TYPE DUT_SourceDataStore :
STRUCT
    {attribute 'pytmc' := 'pv: Valve'}
    fbSourceValve : REFERENCE TO FB_VGC;
    {attribute 'pytmc' := '
        pv: Valid
        io: input
        field: ZNAM Data Invalid
        field: ONAM Data Valid
        field: ZSV MAJOR
        field: OSV NO_ALARM
    '}
    bDataValid : BOOL;

    {attribute 'pytmc' := '
        pv: ChecksOK
        io: input
        field: ZNAM Failed
        field: ONAM Passed
        field: ZSV MAJOR
        field: OSV NO_ALARM
    '}
    bChecksOK : BOOL;
    {attribute 'pytmc' := 'pv: Linear'}
    fbLinear : FB_RangeComparison;
    {attribute 'pytmc' := 'pv: Rotary'}
    fbRotary : FB_RangeComparison;
    {attribute 'pytmc' := 'pv: Goniometer'}
    fbGoniometer : FB_RangeComparison;
    {attribute 'pytmc' := 'pv: NFCenterX'}
    fbNFCentroidX : FB_RangeComparison;
    {attribute 'pytmc' := 'pv: NFCenterY'}
    fbNFCentroidY : FB_RangeComparison;
    {attribute 'pytmc' := 'pv: FFCenterX'}
    fbFFCentroidX : FB_RangeComparison;
    {attribute 'pytmc' := 'pv: FFCenterY'}
    fbFFCentroidY : FB_RangeComparison;
END_STRUCT
END_TYPE

(* stored: Version 1.1.0.1, ProductVersion 3.1.4022.18
   DUT DUT_SourceDataStore: Id {19ae7841-9ce1-47c6-a2ac-e8b660e4994e} *)
